PROPERTY ModuloTurn : dint
GET
ModuloTurn := _Mover.NcToPlc.ModuloSetTurns;
END_GET
END_PROPERTY

PROPERTY Mover : REFERENCE to AXIS_REF
SET
_Mover REF= Mover;
END_SET
END_PROPERTY

PROPERTY MoverId : uint
SET
_nMoverId := MoverId;
END_SET
END_PROPERTY

PROPERTY MoverInfo : REFERENCE to ST_MOVER_INFO
SET


	_stInfo ref= MoverInfo;
END_SET
END_PROPERTY

METHOD MoveToPos : E_PROGRESS
VAR_INPUT
  Execute             : BOOL;
  stMoveData          : ST_MOVE_DATA;
END_VAR
VAR_INST
  _nErrorId           : UDINT;
  _rDelta,
  _rPos               : LREAL;
  _eState             : E_PROGRESS;
END_VAR
IF NOT Execute THEN _eState  := E_PROGRESS.PROGRESS_INIT; END_IF 
IF NOT Check() THEN MoveToPos   := E_PROGRESS.PROGRESS_ERROR; RETURN; END_IF


CASE _eState
OF
  E_PROGRESS.PROGRESS_INIT:
    IF Execute
    THEN
      _nErrorId               := 0;
      _rDelta                 := SEL((stMoveData.rDelta < 0.01), stMoveData.rDelta, 0.05);
      _eState                 := E_PROGRESS.PROGRESS_BUSY;
    END_IF
END_CASE
//-----------------------------------------------------------------------------
//-----------------------------------------------------------------------------
CASE _eState
OF
  E_PROGRESS.PROGRESS_BUSY:
    _eState                   := E_PROGRESS.PROGRESS_PREPARE;
    _fbPower.Override         := stMoveData.rOverride;

    _rPos                     := ABS(_Mover.NcToPlc.ModuloActTurns)* _RailLength + stMoveData.rPos;


    _rLastPosition            := _rPos;
    //_rLastGap                 := stMoveData.rGap;

    _fbMoveAbs(
            Axis              := _Mover, 
            Execute           := FALSE, 
            Position          := _rPos, 
            Velocity          := stMoveData.rVelo, 
            Acceleration      := stMoveData.rAcc, 
            Deceleration      := stMoveData.rAcc, 
            Jerk              := stMoveData.rJerk, 
            BufferMode        := Tc2_MC2.MC_BufferMode.MC_Aborting);

      IF (_eMessageLevel > E_MessageType.eMessageInfo)
      THEN
        _stMsg.eType          := E_MessageType.eMessageVerbose;
        _stMsg.eSubdevice     := e_Subdevice.fbMovePtP;
        _stMsg.iErrorNumber   := _nErrorId;
        _stMsg.sText          := concat(TO_STRING(_eState), ': ');
        _stMsg.sText          := concat(_stMsg.sText, concat('stMoveData.rPos: ', TO_STRING(stMoveData.rPos)));
        f_MessageSet(_stMsg);
      END_IF
END_CASE
//-----------------------------------------------------------------------------
//-----------------------------------------------------------------------------
CASE _eState
OF
  E_PROGRESS.PROGRESS_PREPARE:
    _fbMoveAbs(
            Axis              := _Mover, 
            Execute           := TRUE, 
            Position          := _rPos, 
            Velocity          := stMoveData.rVelo, 
            Acceleration      := stMoveData.rAcc, 
            Deceleration      := stMoveData.rAcc, 
            Jerk              := stMoveData.rJerk, 
            BufferMode        := Tc2_MC2.MC_BufferMode.MC_Aborting);

    IF _fbMoveAbs.Error
    THEN
      _bError                 := TRUE;
      _nErrorId               := _fbMoveAbs.ErrorId;
      _eState                 := E_PROGRESS.PROGRESS_ERROR;

      _stMsg.eType            := E_MessageType.eMessageError;
      _stMsg.eSubdevice       := e_Subdevice.fbMovePtP;
      _stMsg.iErrorNumber     := _nErrorId;
      _stMsg.sText            := TO_STRING(_eState);
      f_MessageSet(_stMsg);

    ELSIF _fbMoveAbs.Active OR 
          _fbMoveAbs.Done
		THEN
      _eState                 := E_PROGRESS.PROGRESS_WORKING;

      IF (_eMessageLevel = E_MessageType.eMessageVerbose)
      THEN
        _stMsg.eType          := E_MessageType.eMessageVerbose;
        _stMsg.eSubdevice     := e_Subdevice.fbMovePtP;
        _stMsg.iErrorNumber   := _nErrorId;
        _stMsg.sText          := concat(TO_STRING(_eState), ': ');
        _stMsg.sText          := concat(_stMsg.sText, '.ModuloActPos: ');
        _stMsg.sText          := concat(_stMsg.sText, TO_STRING(_Mover.NcToPlc.ModuloActPos));
        f_MessageSet(_stMsg);
      END_IF
    END_IF
END_CASE
//-----------------------------------------------------------------------------
//-----------------------------------------------------------------------------
CASE _eState
OF
  E_PROGRESS.PROGRESS_WORKING:
    _fbMoveAbs(
          Axis                := _Mover);

    IF _fbMoveAbs.Error
    THEN
      _bError                 := TRUE;
      _nErrorId               := _fbMoveAbs.ErrorId;
      _stInfo.nErrorId        := _nErrorId;
      _eState                 := E_PROGRESS.PROGRESS_ERROR;

      _stMsg.eType            := E_MessageType.eMessageError;
      _stMsg.eSubdevice       := e_Subdevice.fbMovePtP;
      _stMsg.iErrorNumber     := _nErrorId;
      _stMsg.sText            := TO_STRING(_eState);
      f_MessageSet(_stMsg);

      _fbMoveAbs( 
            Axis              := _Mover, 
            Execute           := FALSE);


    ELSIF (_Mover.NcToPlc.ActPos > _fbMoveAbs.Position - _rDelta) AND
          (_Mover.NcToPlc.ActPos < _fbMoveAbs.Position + _rDelta)
    THEN
      IF NOT _Mover.Status.Moving
      THEN
        _eState               := E_PROGRESS.PROGRESS_DONE;

        IF (_eMessageLevel > E_MessageType.eMessageError)
        THEN
          _stMsg.eType        := E_MessageType.eMessageInfo;
          _stMsg.eSubdevice   := e_Subdevice.fbMovePtP;
          _stMsg.iErrorNumber := _nErrorId;
          _stMsg.sText        := concat(TO_STRING(_eState), ': ');
          _stMsg.sText        := concat(_stMsg.sText, concat('ModActPos: ', TO_STRING(_Mover.NcToPlc.ModuloActPos)));
          f_MessageSet(_stMsg);
        END_IF
      _fbMoveAbs( 
            Axis              := _Mover, 
            Execute           := FALSE);
      END_IF
    END_IF
END_CASE
//-----------------------------------------------------------------------------
//-----------------------------------------------------------------------------

MoveToPos                   := _eState;
END_METHOD

METHOD MoveToPosCa : E_PROGRESS
VAR_INPUT
  Execute             : BOOL;
  stMoveData          : ST_MOVE_DATA;
END_VAR
VAR_INST
  _nErrorId           : UDINT;
  _rDelta,
  _rPos               : LREAL;
  _eState             : E_PROGRESS;
END_VAR
IF NOT Execute THEN _eState  := E_PROGRESS.PROGRESS_INIT; END_IF 
IF NOT Check() THEN MoveToPosCa   := E_PROGRESS.PROGRESS_ERROR; RETURN; END_IF


CASE _eState
OF
  E_PROGRESS.PROGRESS_INIT:
    IF Execute
    THEN
      _nErrorId               := 0;
      _rDelta                 := SEL((stMoveData.rDelta < 0.01), stMoveData.rDelta, 0.05);
      _eState                 := E_PROGRESS.PROGRESS_BUSY;
    END_IF
END_CASE
//-----------------------------------------------------------------------------
//-----------------------------------------------------------------------------
CASE _eState
OF
  E_PROGRESS.PROGRESS_BUSY:
    _eState                   := E_PROGRESS.PROGRESS_PREPARE;
    _fbPower.Override         := stMoveData.rOverride;

    _rPos                     := ABS(_Mover.NcToPlc.ModuloActTurns)* _RailLength + stMoveData.rPos;


    _rLastPosition            := _rPos;
    _rLastGap                 := stMoveData.rGap;

    _fbMoveAbsCa( 
            Axis              := _Mover, 
            Execute           := FALSE, 
            ContinuousUpdate  := TRUE, 
            Position          := _rPos,
            Velocity          := stMoveData.rVelo, 
            Acceleration      := stMoveData.rAcc, 
            Deceleration      := stMoveData.rAcc, 
            Jerk              := stMoveData.rJerk, 
            Gap               := stMoveData.rGap, 
            BufferMode        := Tc3_Mc3Definitions.MC_BUFFER_MODE.mcAborting);

    IF (_eMessageLevel > E_MessageType.eMessageInfo)
    THEN
      _stMsg.eType            := E_MessageType.eMessageVerbose;
      _stMsg.eSubdevice       := e_Subdevice.fbMoveToPosCa;
      _stMsg.iErrorNumber     := _nErrorId;
      _stMsg.sText            := concat(TO_STRING(_eState), ': ');
      _stMsg.sText            := concat(_stMsg.sText, concat('stMoveData.rPos: ', TO_STRING(stMoveData.rPos)));
      f_MessageSet(_stMsg);
    END_IF
END_CASE
//-----------------------------------------------------------------------------
//-----------------------------------------------------------------------------
CASE _eState
OF
  E_PROGRESS.PROGRESS_PREPARE:
    _fbMoveAbsCa( 
            Axis              := _Mover, 
            Execute           := TRUE, 
            ContinuousUpdate  := TRUE, 
            Position          := _rPos,
            Velocity          := stMoveData.rVelo, 
            Acceleration      := stMoveData.rAcc, 
            Deceleration      := stMoveData.rAcc, 
            Jerk              := stMoveData.rJerk, 
            Gap               := stMoveData.rGap, 
            BufferMode        := Tc3_Mc3Definitions.MC_BUFFER_MODE.mcAborting);

    IF _fbMoveAbsCa.Error
    THEN
      _bError                 := TRUE;
      _nErrorId               := _fbMoveAbsCa.ErrorId;
      _stInfo.nErrorId        := _nErrorId;
      _eState                 := E_PROGRESS.PROGRESS_ERROR;

      _stMsg.eType            := E_MessageType.eMessageError;
      _stMsg.eSubdevice       := e_Subdevice.fbMoveToPosCa;
      _stMsg.iErrorNumber     := _nErrorId;
      _stMsg.sText            := TO_STRING(_eState);
      f_MessageSet(_stMsg);

    ELSIF _fbMoveAbsCa.Active OR 
          _fbMoveAbsCa.Done
		THEN
      _eState                 := E_PROGRESS.PROGRESS_WORKING;

      IF (_eMessageLevel = E_MessageType.eMessageVerbose)
      THEN
        _stMsg.eType          := E_MessageType.eMessageVerbose;
        _stMsg.eSubdevice     := e_Subdevice.fbMoveToPosCa;
        _stMsg.iErrorNumber   := _nErrorId;
        _stMsg.sText          := concat(TO_STRING(_eState), ': ');
        _stMsg.sText          := concat(_stMsg.sText, '.ModuloActPos: ');
        _stMsg.sText          := concat(_stMsg.sText, TO_STRING(_Mover.NcToPlc.ModuloActPos));
        f_MessageSet(_stMsg);
      END_IF
    END_IF
END_CASE
//-----------------------------------------------------------------------------
//-----------------------------------------------------------------------------
CASE _eState
OF
  E_PROGRESS.PROGRESS_WORKING:
    _fbMoveAbsCa(
          Axis                := _Mover);

    IF _fbMoveAbsCa.Error
    THEN
      _bError                 := TRUE;
      _nErrorId               := _fbMoveAbsCa.ErrorId;
      _stInfo.nErrorId        := _nErrorId;
      _fbMoveAbsCa( 
            Axis              := _Mover, 
            Execute           := FALSE);

      _eState                 := E_PROGRESS.PROGRESS_ERROR;

      _stMsg.eType            := E_MessageType.eMessageError;
      _stMsg.eSubdevice       := e_Subdevice.fbMoveToPosCa;
      _stMsg.iErrorNumber     := _nErrorId;
      _stMsg.sText            := concat(TO_STRING(_eState), ': ');
      _stMsg.sText            := concat(_stMsg.sText, concat('ModActPos: ', TO_STRING(_Mover.NcToPlc.ModuloActPos)));

      f_MessageSet(_stMsg);

    ELSIF (_Mover.NcToPlc.ActPos > _fbMoveAbsCa.Position - _rDelta) AND
          (_Mover.NcToPlc.ActPos < _fbMoveAbsCa.Position + _rDelta)
    THEN
      IF NOT _Mover.Status.Moving
      THEN
        _eState               := E_PROGRESS.PROGRESS_DONE;

        IF (_eMessageLevel > E_MessageType.eMessageError)
        THEN
          _stMsg.eType        := E_MessageType.eMessageInfo;
          _stMsg.eSubdevice   := e_Subdevice.fbMoveToPosCa;
          _stMsg.iErrorNumber := _nErrorId;
          _stMsg.sText        := concat(TO_STRING(_eState), ': ');
          _stMsg.sText        := concat(_stMsg.sText, concat('ModActPos: ', TO_STRING(_Mover.NcToPlc.ModuloActPos)));
          f_MessageSet(_stMsg);
        END_IF
      _fbMoveAbsCa( 
            Axis              := _Mover, 
            Execute           := FALSE);
      END_IF
    END_IF
END_CASE
//-----------------------------------------------------------------------------
//-----------------------------------------------------------------------------

MoveToPosCa                   := _eState;
END_METHOD

PROPERTY RailLength : LREAL
GET
RailLength := _RailLength;
END_GET
SET
_RailLength := RailLength;
END_SET
END_PROPERTY

METHOD Reset : E_PROGRESS
VAR_INPUT
  Execute             : BOOL;
END_VAR
VAR_INST
  _nErrorId           : UDINT;
  _eState             : E_PROGRESS;
END_VAR
IF NOT Execute THEN _eState  := E_PROGRESS.PROGRESS_INIT; END_IF 
IF NOT Check() THEN Reset    := E_PROGRESS.PROGRESS_ERROR; RETURN; END_IF


CASE _eState
OF
  E_PROGRESS.PROGRESS_INIT:
    IF Execute
    THEN
      _stInfo.nErrorId        :=
      _nErrorId               := 0;
      _eState                 := E_PROGRESS.PROGRESS_BUSY;
    END_IF
END_CASE
//-----------------------------------------------------------------------------
//-----------------------------------------------------------------------------
CASE _eState
OF
  E_PROGRESS.PROGRESS_BUSY:
    _eState                   := E_PROGRESS.PROGRESS_PREPARE;
    _fbReset(
            Axis              := _Mover, 
            Execute           := FALSE);

    IF (_eMessageLevel > E_MessageType.eMessageInfo)
    THEN
      _stMsg.eType            := E_MessageType.eMessageVerbose;
      _stMsg.eSubdevice       := e_Subdevice.fbReset;
      _stMsg.iErrorNumber     := _nErrorId;
      _stMsg.sText            := TO_STRING(_eState);
      f_MessageSet(_stMsg);
    END_IF
END_CASE
//-----------------------------------------------------------------------------
//-----------------------------------------------------------------------------
CASE _eState
OF
  E_PROGRESS.PROGRESS_PREPARE:
    _fbReset(
            Axis              := _Mover, 
            Execute           := TRUE);

    IF _fbReset.Error
    THEN
      _nErrorId               := _fbReset.ErrorID;
      _eState                 := E_PROGRESS.PROGRESS_ERROR;

      _stMsg.eType            := E_MessageType.eMessageError;
      _stMsg.eSubdevice       := e_Subdevice.fbReset;
      _stMsg.iErrorNumber     := _nErrorId;
      _stMsg.sText            := TO_STRING(_eState);
      f_MessageSet(_stMsg);

    ELSIF NOT _Mover.Status.Moving
    THEN
      _eState                 := E_PROGRESS.PROGRESS_DONE;

      IF (_eMessageLevel > E_MessageType.eMessageError)
      THEN
        _stMsg.eType          := E_MessageType.eMessageInfo;
        _stMsg.eSubdevice     := e_Subdevice.fbReset;
        _stMsg.iErrorNumber   := _nErrorId;
        _stMsg.sText          := TO_STRING(_eState);
        f_MessageSet(_stMsg);
      END_IF
    END_IF
END_CASE
//-----------------------------------------------------------------------------
//-----------------------------------------------------------------------------
CASE _eState
OF
  E_PROGRESS.PROGRESS_ERROR,
  E_PROGRESS.PROGRESS_DONE:
    _stInfo.nErrorId          := _nErrorId;
    _fbReset(
            Axis              := _Mover, 
            Execute           := FALSE);
			
	_bError := FALSE;		
END_CASE
//-----------------------------------------------------------------------------
//-----------------------------------------------------------------------------

Reset                         := _eState;
END_METHOD

METHOD SendToAbsPosCa : E_PROGRESS
VAR_INPUT
  Execute             : BOOL;
  stMoveData          : ST_MOVE_DATA;
END_VAR
VAR_INST
  _nErrorId           : UDINT;
  _rPos               : LREAL;
  _rStart             : LREAL;
  _eState             : E_PROGRESS;
END_VAR
IF NOT Execute THEN _eState  := E_PROGRESS.PROGRESS_INIT; END_IF 
IF NOT Check() THEN SendToAbsPosCa   := E_PROGRESS.PROGRESS_ERROR; RETURN; END_IF


CASE _eState
OF
  E_PROGRESS.PROGRESS_INIT:
    IF Execute
    THEN
      _nErrorId               := 0;
      _rStart                 := _Mover.NcToPlc.ActPos;

      _eState                 := E_PROGRESS.PROGRESS_BUSY;
    END_IF
END_CASE
//-----------------------------------------------------------------------------
//-----------------------------------------------------------------------------
CASE _eState
OF
  E_PROGRESS.PROGRESS_BUSY:
    _eState                   := E_PROGRESS.PROGRESS_PREPARE;
    _fbPower.Override         := stMoveData.rOverride;

    _rPos                     := stMoveData.rPos;
	
    _rLastPosition            := _rPos;
    _rLastGap                 := stMoveData.rGap;

    _fbMoveAbsCa( 
            Axis              := _Mover, 
            Execute           := FALSE, 
            ContinuousUpdate  := TRUE, 
            Position          := _rPos,
            Velocity          := stMoveData.rVelo, 
            Acceleration      := stMoveData.rAcc, 
            Deceleration      := stMoveData.rAcc, 
            Jerk              := stMoveData.rJerk, 
            Gap               := stMoveData.rGap, 
            BufferMode        := Tc3_Mc3Definitions.MC_BUFFER_MODE.mcAborting);

    IF (_eMessageLevel > E_MessageType.eMessageVerbose)
    THEN
      _stMsg.eType            := E_MessageType.eMessageSentient;
      _stMsg.eSubdevice       := e_Subdevice.fbSendToAbsPosCa;
      _stMsg.iErrorNumber     := _nErrorId;
      _stMsg.sText            := concat(TO_STRING(_eState), ': ');
      _stMsg.sText            := concat(_stMsg.sText, 'stMoveData.rPos: ');
      _stMsg.sText            := concat(_stMsg.sText, TO_STRING(stMoveData.rPos));
      f_MessageSet(_stMsg);

      _stMsg.eType            := E_MessageType.eMessageSentient;
      _stMsg.eSubdevice       := e_Subdevice.fbSendToAbsPosCa;
      _stMsg.iErrorNumber     := _nErrorId;
      _stMsg.sText            := concat(TO_STRING(_eState), ': ');
      _stMsg.sText            := concat(_stMsg.sText, '.rDistance: ');
      _stMsg.sText            := concat(_stMsg.sText, TO_STRING(stMoveData.rDistance));
      f_MessageSet(_stMsg);
    END_IF
END_CASE
//-----------------------------------------------------------------------------
//-----------------------------------------------------------------------------
CASE _eState
OF
  E_PROGRESS.PROGRESS_PREPARE:
    _fbMoveAbsCa( 
            Axis              := _Mover, 
            Execute           := TRUE, 
            ContinuousUpdate  := TRUE, 
            Position          := _rPos,
            Velocity          := stMoveData.rVelo, 
            Acceleration      := stMoveData.rAcc, 
            Deceleration      := stMoveData.rAcc, 
            Jerk              := stMoveData.rJerk, 
            Gap               := stMoveData.rGap, 
            BufferMode        := Tc3_Mc3Definitions.MC_BUFFER_MODE.mcAborting);

    IF _fbMoveAbsCa.Error
    THEN
      _bError                 := TRUE;
      _nErrorId               := _fbMoveAbsCa.ErrorId;
      _stInfo.nErrorId        := _nErrorId;
      _eState                 := E_PROGRESS.PROGRESS_ERROR;

      _stMsg.eType            := E_MessageType.eMessageError;
      _stMsg.eSubdevice       := e_Subdevice.fbSendToAbsPosCa;
      _stMsg.iErrorNumber     := _nErrorId;
      _stMsg.sText            := TO_STRING(_eState);
      f_MessageSet(_stMsg);

    ELSIF _fbMoveAbsCa.Active OR
          _fbMoveAbsCa.Done
    THEN
      _eState                 := E_PROGRESS.PROGRESS_WORKING;

      IF (_eMessageLevel > E_MessageType.eMessageVerbose)
      THEN
        _stMsg.eType          := E_MessageType.eMessageSentient;
        _stMsg.eSubdevice     := e_Subdevice.fbSendToAbsPosCa;
        _stMsg.iErrorNumber   := _nErrorId;
        _stMsg.sText          := concat(TO_STRING(_eState), ': ');
        _stMsg.sText          := concat(_stMsg.sText, '.ActPos: ');
        _stMsg.sText          := concat(_stMsg.sText, TO_STRING(_Mover.NcToPlc.ActPos));
        //f_MessageSet(_stMsg);
      END_IF
    END_IF
END_CASE
//-----------------------------------------------------------------------------
//-----------------------------------------------------------------------------
CASE _eState
OF
  E_PROGRESS.PROGRESS_WORKING:
    _fbMoveAbsCa(
            Axis              := _Mover);

    IF _fbMoveAbsCa.Error
    THEN
      _bError                 := TRUE;
      _nErrorId               := _fbMoveAbsCa.ErrorId;
      _stInfo.nErrorId        := _nErrorId;
      _fbMoveAbsCa( 
            Axis              := _Mover, 
            Execute           := FALSE);

      _eState                 := E_PROGRESS.PROGRESS_ERROR;

      _stMsg.eType            := E_MessageType.eMessageError;
      _stMsg.eSubdevice       := e_Subdevice.fbSendToAbsPosCa;
      _stMsg.iErrorNumber     := _nErrorId;
      _stMsg.sText            := TO_STRING(_eState);
      f_MessageSet(_stMsg);

    ELSIF (_Mover.NcToPlc.ActPos > _rStart + stMoveData.rDistance)
    THEN
      _eState                 := E_PROGRESS.PROGRESS_DONE;

      IF (_eMessageLevel > E_MessageType.eMessageError)
      THEN
        _stMsg.eType          := E_MessageType.eMessageInfo;
        _stMsg.eSubdevice     := e_Subdevice.fbSendToAbsPosCa;
        _stMsg.iErrorNumber   := _nErrorId;
        _stMsg.sText          := concat(TO_STRING(_eState), ': ');
        _stMsg.sText          := concat(_stMsg.sText, '.ActPos: ');
        _stMsg.sText          := concat(_stMsg.sText, TO_STRING(_Mover.NcToPlc.ActPos));
        _stMsg.sText          := concat(_stMsg.sText, ' ');
        _stMsg.sText          := concat(_stMsg.sText, '.ActVelo: ');
        _stMsg.sText          := concat(_stMsg.sText, TO_STRING(_Mover.NcToPlc.ActVelo));

        f_MessageSet(_stMsg);
      END_IF
      _fbMoveAbsCa( 
            Axis              := _Mover, 
            Execute           := FALSE);
    END_IF
END_CASE
//-----------------------------------------------------------------------------
//-----------------------------------------------------------------------------

SendToAbsPosCa                := _eState;
END_METHOD

METHOD SendToModuloPosCa : E_PROGRESS
VAR_INPUT
  Execute             : BOOL;
  stMoveData          : ST_MOVE_DATA;
END_VAR
VAR_INST
  _nErrorId           : UDINT;
  _rPos               : LREAL;
  _rStart             : LREAL;
  _eState             : E_PROGRESS;
END_VAR
IF NOT Execute THEN _eState  := E_PROGRESS.PROGRESS_INIT; END_IF 
IF NOT Check() THEN SendToModuloPosCa   := E_PROGRESS.PROGRESS_ERROR; RETURN; END_IF


CASE _eState
OF
  E_PROGRESS.PROGRESS_INIT:
    IF Execute
    THEN
      _nErrorId               := 0;
      _rStart                 := _Mover.NcToPlc.ActPos;

      _eState                 := E_PROGRESS.PROGRESS_BUSY;
    END_IF
    _fbMoveAbsCa( 
          Axis              := _Mover, 
          Execute           := FALSE);
END_CASE
//-----------------------------------------------------------------------------
//-----------------------------------------------------------------------------
CASE _eState
OF
  E_PROGRESS.PROGRESS_BUSY:
    _eState                   := E_PROGRESS.PROGRESS_PREPARE;
    _fbPower.Override         := stMoveData.rOverride;

    _rPos                     := ABS(_Mover.NcToPlc.ModuloActTurns)* _RailLength + stMoveData.rPos;
	
    _rLastPosition            := _rPos;
    _rLastGap                 := stMoveData.rGap;

    _fbMoveAbsCa( 
            Axis              := _Mover, 
            Execute           := FALSE, 
            ContinuousUpdate  := TRUE, 
            Position          := _rPos,
            Velocity          := stMoveData.rVelo, 
            Acceleration      := stMoveData.rAcc, 
            Deceleration      := stMoveData.rAcc, 
            Jerk              := stMoveData.rJerk, 
            Gap               := stMoveData.rGap, 
            BufferMode        := Tc3_Mc3Definitions.MC_BUFFER_MODE.mcAborting);

    IF (_eMessageLevel > E_MessageType.eMessageVerbose)
    THEN
      _stMsg.eType            := E_MessageType.eMessageSentient;
      _stMsg.eSubdevice       := e_Subdevice.fbSendToModuloPosCa;
      _stMsg.iErrorNumber     := _nErrorId;
      _stMsg.sText            := concat(TO_STRING(_eState), ': ');
      _stMsg.sText            := concat(_stMsg.sText, 'stMoveData.rPos: ');
      _stMsg.sText            := concat(_stMsg.sText, TO_STRING(stMoveData.rPos));
      f_MessageSet(_stMsg);

      _stMsg.eType            := E_MessageType.eMessageSentient;
      _stMsg.eSubdevice       := e_Subdevice.fbSendToModuloPosCa;
      _stMsg.iErrorNumber     := _nErrorId;
      _stMsg.sText            := concat(TO_STRING(_eState), ': ');
      _stMsg.sText            := concat(_stMsg.sText, '.rDistance: ');
      _stMsg.sText            := concat(_stMsg.sText, TO_STRING(stMoveData.rDistance));
      f_MessageSet(_stMsg);

    END_IF
END_CASE
//-----------------------------------------------------------------------------
//-----------------------------------------------------------------------------
CASE _eState
OF
  E_PROGRESS.PROGRESS_PREPARE:
    _fbMoveAbsCa( 
            Axis              := _Mover, 
            Execute           := TRUE, 
            ContinuousUpdate  := TRUE, 
            Position          := _rPos,
            Velocity          := stMoveData.rVelo, 
            Acceleration      := stMoveData.rAcc, 
            Deceleration      := stMoveData.rAcc, 
            Jerk              := stMoveData.rJerk, 
            Gap               := stMoveData.rGap, 
            BufferMode        := Tc3_Mc3Definitions.MC_BUFFER_MODE.mcAborting);

    IF _fbMoveAbsCa.Error
    THEN
      _bError                 := TRUE;
      _nErrorId               := _fbMoveAbsCa.ErrorId;
      _stInfo.nErrorId        := _nErrorId;
      _eState                 := E_PROGRESS.PROGRESS_ERROR;

      _stMsg.eType            := E_MessageType.eMessageError;
      _stMsg.eSubdevice       := e_Subdevice.fbSendToModuloPosCa;
      _stMsg.iErrorNumber     := _nErrorId;
      _stMsg.sText            := TO_STRING(_eState);
      f_MessageSet(_stMsg);

      _fbMoveAbsCa( 
            Axis              := _Mover, 
            Execute           := FALSE);

    ELSIF _fbMoveAbsCa.Active OR
          _fbMoveAbsCa.Done
    THEN
      _eState                 := E_PROGRESS.PROGRESS_WORKING;

      IF (_eMessageLevel > E_MessageType.eMessageVerbose)
      THEN
        _stMsg.eType          := E_MessageType.eMessageSentient;
        _stMsg.eSubdevice     := e_Subdevice.fbSendToModuloPosCa;
        _stMsg.iErrorNumber   := _nErrorId;
        _stMsg.sText            := concat(TO_STRING(_eState), ': ');
        _stMsg.sText          := concat(_stMsg.sText, '.ModuloActPos: ');
        _stMsg.sText          := concat(_stMsg.sText, TO_STRING(_Mover.NcToPlc.ModuloActPos));
        //f_MessageSet(_stMsg);
      END_IF
(*
    ELSIF (_Mover.NcToPlc.ActPos > _rStart + stMoveData.rDistance)
    THEN
      _eState                 := E_PROGRESS.PROGRESS_DONE;

      IF (_eMessageLevel < E_MessageType.eMessageError)
      THEN
        _stMsg.eType          := E_MessageType.eMessageInfo;
        _stMsg.eSubdevice     := e_Subdevice.fbSendToModuloPosCa;
        _stMsg.iErrorNumber   := _nErrorId;
        _stMsg.sText          := TO_STRING(_eState);
        f_MessageSet(_stMsg);
      END_IF
      _fbMoveAbsCa( 
            Axis              := _Mover, 
            Execute           := FALSE);
*)
    END_IF
END_CASE
//-----------------------------------------------------------------------------
//-----------------------------------------------------------------------------
CASE _eState
OF
  E_PROGRESS.PROGRESS_WORKING:
    _fbMoveAbsCa(
            Axis              := _Mover);

    IF _fbMoveAbsCa.Error
    THEN
      _bError                 := TRUE;
      _nErrorId               := _fbMoveAbsCa.ErrorId;
      _stInfo.nErrorId        := _nErrorId;
      _fbMoveAbsCa( 
            Axis              := _Mover, 
            Execute           := FALSE);

      _eState                 := E_PROGRESS.PROGRESS_ERROR;

      _stMsg.eType            := E_MessageType.eMessageError;
      _stMsg.eSubdevice       := e_Subdevice.fbSendToModuloPosCa;
      _stMsg.iErrorNumber     := _nErrorId;
      _stMsg.sText            := TO_STRING(_eState);
      f_MessageSet(_stMsg);

    ELSIF (_Mover.NcToPlc.ActPos > _rStart + stMoveData.rDistance)
    THEN
      _eState                 := E_PROGRESS.PROGRESS_DONE;

      IF (_eMessageLevel > E_MessageType.eMessageError)
      THEN
        _stMsg.eType          := E_MessageType.eMessageInfo;
        _stMsg.eSubdevice     := e_Subdevice.fbSendToModuloPosCa;
        _stMsg.iErrorNumber   := _nErrorId;
        _stMsg.sText          := concat(TO_STRING(_eState), ': ');
        _stMsg.sText          := concat(_stMsg.sText, '.ModuloActPos: ');
        _stMsg.sText          := concat(_stMsg.sText, TO_STRING(_Mover.NcToPlc.ModuloActPos));
        _stMsg.sText          := concat(_stMsg.sText, ' ');
        _stMsg.sText          := concat(_stMsg.sText, '.ActVelo: ');
        _stMsg.sText          := concat(_stMsg.sText, TO_STRING(_Mover.NcToPlc.ActVelo));
        f_MessageSet(_stMsg);
      END_IF
      _fbMoveAbsCa( 
            Axis              := _Mover, 
            Execute           := FALSE);
    END_IF
END_CASE
//-----------------------------------------------------------------------------
//-----------------------------------------------------------------------------

SendToModuloPosCa                   := _eState;
END_METHOD

METHOD Stop : E_PROGRESS
VAR_INPUT
  Execute             : BOOL;
  stMoveData          : ST_MOVE_DATA;
END_VAR
VAR_INST
  _nErrorId           : UDINT;
  _eState             : E_PROGRESS;
END_VAR
IF NOT Execute 
THEN 
	_eState := E_PROGRESS.PROGRESS_INIT; 
END_IF 
IF NOT Check() 
THEN 
	Stop := E_PROGRESS.PROGRESS_ERROR; 
	RETURN; 
END_IF


CASE _eState
OF
  E_PROGRESS.PROGRESS_INIT:
    IF Execute
    THEN
      _nErrorId               := 0;
      _eState                 := E_PROGRESS.PROGRESS_BUSY;
    END_IF
END_CASE
//-----------------------------------------------------------------------------
//-----------------------------------------------------------------------------
CASE _eState
OF
  E_PROGRESS.PROGRESS_BUSY:
    _eState                   := E_PROGRESS.PROGRESS_PREPARE;
    _fbStop(
            Axis              := _Mover, 
            Execute           := FALSE, 
            Deceleration      := stMoveData.rAcc, 
            Jerk              := stMoveData.rJerk); 

    IF (_eMessageLevel > E_MessageType.eMessageInfo)
    THEN
      _stMsg.eType            := E_MessageType.eMessageVerbose;
      _stMsg.eSubdevice       := e_Subdevice.fbStop;
      _stMsg.iErrorNumber     := _nErrorId;
      _stMsg.sText            := TO_STRING(_eState);
      f_MessageSet(_stMsg);
    END_IF
END_CASE
//-----------------------------------------------------------------------------
//-----------------------------------------------------------------------------
CASE _eState
OF
  E_PROGRESS.PROGRESS_PREPARE:
    _fbStop(Axis              := _Mover, 
            Execute           := TRUE, 
            Deceleration      := stMoveData.rAcc, 
            Jerk              := stMoveData.rJerk);

    IF _fbStop.Error
    THEN
      _bError                 := TRUE;
      _nErrorId               := _fbStop.ErrorID;
      _eState                 := E_PROGRESS.PROGRESS_ERROR;

      _stMsg.eType            := E_MessageType.eMessageError;
      _stMsg.eSubdevice       := e_Subdevice.fbStop;
      _stMsg.iErrorNumber     := _nErrorId;
      _stMsg.sText            := TO_STRING(_eState);
      f_MessageSet(_stMsg);

    ELSIF _fbStop.Done
    THEN
      _eState                 := E_PROGRESS.PROGRESS_DONE;

      IF (_eMessageLevel > E_MessageType.eMessageError)
      THEN
        _stMsg.eType          := E_MessageType.eMessageInfo;
        _stMsg.eSubdevice     := e_Subdevice.fbStop;
        _stMsg.iErrorNumber   := _nErrorId;
        _stMsg.sText          := TO_STRING(_eState);
        f_MessageSet(_stMsg);
      END_IF
    END_IF
END_CASE
//-----------------------------------------------------------------------------
//-----------------------------------------------------------------------------
CASE _eState
OF
  E_PROGRESS.PROGRESS_ERROR,
  E_PROGRESS.PROGRESS_DONE:
    _stInfo.nErrorId          := _nErrorId;
    _fbStop(
            Axis              := _Mover, 
            Execute           := FALSE);
END_CASE
//-----------------------------------------------------------------------------
//-----------------------------------------------------------------------------

Stop                          := _eState;
END_METHOD

END_FUNCTION_BLOCK

// ---- APPLICATION/_types/Initialization_Robot.TcPOU
FUNCTION Initialization_Robot : BOOL
VAR_INPUT
END_VAR
VAR
  _nBufferOutfeedTarget       : ARRAY[1..2] OF E_INSTANCE;
  _nStnFrst                   : UINT;
END_VAR

//*************************************************************************************************************
//
// build configuration for Instances and ProcessInterfaces
//
//*************************************************************************************************************
//*************************************************************************************************************
// - ProcessConductor : Instance with connection to a cyclic linked list 
//                      Here does The Ticket with target processId and bitmask arrive 
//                      this instance forwards the ticket to its destination
//                        destination is BufferInfeed
//-------------------------------------------------------------------------------------------------------------
// whoami
//
// ticket box - transfersystem drops ticket
//-------------------------------------------------------------------------------------------------------------
ProcessConductor.ProcessId                := ProcessCollector[E_INSTANCE.PROCESS_CONDUCTOR].ProcessId;
ProcessConductor.CollectorInterface       := ItfProcessCollector;
ProcessConductor.ProcessLinkedLists       := ItfProcessList;

//*************************************************************************************************************
// - BufferInfeed     : single XtsStation which looks for input trigger from transfersystem, 
//                      transfersystem writes positions of XtsStations to be used at Infeed. 
//                      BufferInfeed is writing ItfProcessCollector[BufferInfeed.ProcessTarget].ActivateStation 
//                        for BufferInfeed target (Infeed / 12 XtsStations).
//                      BufferInfeed sends required amount of movers to WaitPos of XtsStations 
//                        of BufferInfeed target (Infeed / 12 XtsStations).
//-------------------------------------------------------------------------------------------------------------
// whoami
//
// process target (Infeed / 12 XtsStations)
//-------------------------------------------------------------------------------------------------------------
BufferInfeed.ProcessId                    := ProcessCollector[E_INSTANCE.BUFFER_INFEED].ProcessId;
BufferInfeed.ProcessTarget                := ProcessCollector[E_INSTANCE.INFEED].ProcessId;
BufferInfeed.CollectorInterface           := ItfProcessCollector;
BufferInfeed.ProcessLinkedLists           := ItfProcessList;
//-------------------------------------------------------------------------------------------------------------
// configure range of XtsStations for process
//
// see MAIN.StationParameterInit() for positions and dyn constraints
//-------------------------------------------------------------------------------------------------------------
ItfProcessCollector[BufferInfeed.ProcessId].StationFirst  := 53;
ItfProcessCollector[BufferInfeed.ProcessId].StationLast   := 53;

_nStnFrst                                 := ProcessCollector[BufferInfeed.ProcessId].StationFirst;
BufferInfeed.CheckPosition                := 15.0;

//-------------------------------------------------------------------------------------------------------------
//-------------------------------------------------------------------------------------------------------------
//*************************************************************************************************************
//*************************************************************************************************************
// - Infeed         : 12 XtsStations for transfersystem to unload
//                    Infeed is pulling in the movers according to list entry from BufferInfeed
//                    one stop only
//                    must be checked for all mover standstill in PosStop[1] of each XtsStation
//                    must be released by handshake from transfersystem (this is done by a TON for now)
//-------------------------------------------------------------------------------------------------------------
// whoami
//
// process target (BufferOutfeed / 1 XtsStation)
// TODO: 
//    configure infeed target for OUTFEED_CLAMP (12 XtsStations)
//    Infeed.ProcessTarget  := ProcessCollector[E_INSTANCE.OUTFEED_CLAMP].ProcessId;
//-------------------------------------------------------------------------------------------------------------
Infeed.ProcessId                          := ProcessCollector[E_INSTANCE.INFEED].ProcessId;
Infeed.ProcessTarget                      := ProcessCollector[E_INSTANCE.BUFFER_OUTFEED].ProcessId;
Infeed.CollectorInterface                 := ItfProcessCollector;
Infeed.ProcessLinkedLists                 := ItfProcessList;
//-------------------------------------------------------------------------------------------------------------
// configure range of XtsStations for process
//
// see MAIN.StationParameterInit() for positions and dyn constraints
//-------------------------------------------------------------------------------------------------------------
ItfProcessCollector[Infeed.ProcessId].StationFirst        :=  1;
ItfProcessCollector[Infeed.ProcessId].StationLast         := 12;
//-------------------------------------------------------------------------------------------------------------
//-------------------------------------------------------------------------------------------------------------
//*************************************************************************************************************
//*************************************************************************************************************
// - BufferOutfeed  : single XtsStation which distributes movers to specified range 
//                    Infeed sends all movers here 
//                    BufferOutfeed ensures that OutputR2 and OutputR1 have 12 movers each for every job
//                    BufferOutfeed checks if the Queue of this single XtsStation is empty or not
//-------------------------------------------------------------------------------------------------------------
// whoami
//
// process target (Outfeed (OutfeedR2 & OutfeedR1) / 24 XtsStations)
//
//  - optional process target (Outfeed 12 XtsStations)
//-------------------------------------------------------------------------------------------------------------
_nBufferOutfeedTarget[1] := E_INSTANCE.OUTFEED_ROBOT_R1;
_nBufferOutfeedTarget[2] := E_INSTANCE.OUTFEED_ROBOT_R2;

BufferOutfeed.ProcessId              := E_INSTANCE.BUFFER_OUTFEED;
BufferOutfeed.ProcessTarget          := _nBufferOutfeedTarget; 
BufferOutfeed.CollectorInterface     := ItfProcessCollector;
BufferOutfeed.ProcessLinkedLists     := ItfProcessList;
//-------------------------------------------------------------------------------------------------------------
// configure range of XtsStations for process
//
// see MAIN.StationParameterInit() for positions and dyn constraints
//-------------------------------------------------------------------------------------------------------------
ItfProcessCollector[BufferOutfeed.ProcessId].StationFirst  := 25;
ItfProcessCollector[BufferOutfeed.ProcessId].StationLast   := 25;

_nStnFrst                                 := ProcessCollector[BufferOutfeed.ProcessId].StationFirst;
BufferOutfeed.CheckPosition          := 2500.0;
//-------------------------------------------------------------------------------------------------------------
//-------------------------------------------------------------------------------------------------------------
//*************************************************************************************************************
//*************************************************************************************************************
// - Outfeed_R1  : 12 XtsStations for Robot 
//                    All XtsStations must be filled before robot can start 
//                    affter process all movers are sent to Sender process (high speed for the way back)
//                     
//                    
//-------------------------------------------------------------------------------------------------------------
// whoami
//
// process target (SenderFast / 1 XtsStation)
//-------------------------------------------------------------------------------------------------------------
Outfeed_R1.ProcessId                      := E_INSTANCE.OUTFEED_ROBOT_R1;
Outfeed_R1.ProcessTarget                  := ProcessCollector[E_INSTANCE.SENDER_FAST].ProcessId;
Outfeed_R1.CollectorInterface             := ItfProcessCollector;
Outfeed_R1.ProcessLinkedLists             := ItfProcessList;
//-------------------------------------------------------------------------------------------------------------
// configure range of XtsStations for process
//
// see MAIN.StationParameterInit() for positions and dyn constraints
//-------------------------------------------------------------------------------------------------------------
ItfProcessCollector[Outfeed_R1.ProcessId].StationFirst  := 26;
ItfProcessCollector[Outfeed_R1.ProcessId].StationLast   := 37;

_nStnFrst                                 := ProcessCollector[Outfeed_R1.ProcessId].StationFirst;
Outfeed_R1.CheckPosition                  := 6000.0;
//-------------------------------------------------------------------------------------------------------------
//-------------------------------------------------------------------------------------------------------------
//*************************************************************************************************************
//*************************************************************************************************************
// - Outfeed_R2  : 12 XtsStations for Robot 
//                    All XtsStations must be filled before robot can start 
//                    affter process all movers are sent to Sender process (high speed for the way back)
//                     
//                    
//-------------------------------------------------------------------------------------------------------------
// whoami
//
// process target (SenderFast / 1 XtsStation)
//-------------------------------------------------------------------------------------------------------------
Outfeed_R2.ProcessId                      := E_INSTANCE.OUTFEED_ROBOT_R2;
Outfeed_R2.ProcessTarget                  := ProcessCollector[E_INSTANCE.SENDER_FAST].ProcessId;
Outfeed_R2.CollectorInterface             := ItfProcessCollector;
Outfeed_R2.ProcessLinkedLists             := ItfProcessList;
//-------------------------------------------------------------------------------------------------------------
// configure range of XtsStations for process
//
// see MAIN.StationParameterInit() for positions and dyn constraints
//-------------------------------------------------------------------------------------------------------------
ItfProcessCollector[Outfeed_R2.ProcessId].StationFirst  := 38;
ItfProcessCollector[Outfeed_R2.ProcessId].StationLast   := 49;

_nStnFrst                                 := ProcessCollector[Outfeed_R2.ProcessId].StationFirst;
Outfeed_R2.CheckPosition                  := 6000.0;
//-------------------------------------------------------------------------------------------------------------
//-------------------------------------------------------------------------------------------------------------
//*************************************************************************************************************
//*************************************************************************************************************
// - SenderFast  : 1 XtsStation 
//                    movers are handled when entering position area 
//                    movers are accelerated to max speed
//                    movers do not stop here
//                    
//-------------------------------------------------------------------------------------------------------------
// whoami
//
// process target (SenderBufferInfeed / 1 XtsStation)
//-------------------------------------------------------------------------------------------------------------
SenderFast.ProcessId                      := E_INSTANCE.SENDER_FAST;
SenderFast.ProcessTarget                  := ProcessCollector[E_INSTANCE.SENDER_BUFFER_INFEED].ProcessId;
SenderFast.CollectorInterface             := ItfProcessCollector;
SenderFast.ProcessLinkedLists             := ItfProcessList;
//-------------------------------------------------------------------------------------------------------------
// configure range of XtsStations for process
//
// see MAIN.StationParameterInit() for positions and dyn constraints
//-------------------------------------------------------------------------------------------------------------
ItfProcessCollector[SenderFast.ProcessId].StationFirst  := 51;
ItfProcessCollector[SenderFast.ProcessId].StationLast   := 51;

_nStnFrst                                 := ProcessCollector[SenderFast.ProcessId].StationFirst;
SenderFast.CheckPosition                  := GVL_XTS.StationParameter[_nStnFrst].rPosWait - 500.0;
//-------------------------------------------------------------------------------------------------------------
//-------------------------------------------------------------------------------------------------------------
//*************************************************************************************************************
//*************************************************************************************************************
// - SenderBufferInfeed  : 1 XtsStation 
//                    movers are handled when entering position area 
//                    movers are sent to BufferInfeed, so that BufferInfeed has 12 mover ready
//                    movers do stop here, wait until there is room for movers
//                    
//-------------------------------------------------------------------------------------------------------------
// whoami
//
// process target (SenderBufferInfeed / 1 XtsStation)
//-------------------------------------------------------------------------------------------------------------
SenderBufferInfeed.ProcessId              := E_INSTANCE.SENDER_BUFFER_INFEED;
SenderBufferInfeed.ProcessTarget          := ProcessCollector[E_INSTANCE.BUFFER_INFEED].ProcessId;
SenderBufferInfeed.CollectorInterface     := ItfProcessCollector;
SenderBufferInfeed.ProcessLinkedLists     := ItfProcessList;
//-------------------------------------------------------------------------------------------------------------
// configure range of XtsStations for process
//
// see MAIN.StationParameterInit() for positions and dyn constraints
//-------------------------------------------------------------------------------------------------------------
ItfProcessCollector[SenderBufferInfeed.ProcessId].StationFirst  := 52;
ItfProcessCollector[SenderBufferInfeed.ProcessId].StationLast   := 52;

_nStnFrst                                 := ProcessCollector[SenderBufferInfeed.ProcessId].StationFirst;
SenderBufferInfeed.CheckPosition          := GVL_XTS.StationParameter[_nStnFrst].rPosWait - 1250.0;
//-------------------------------------------------------------------------------------------------------------
//-------------------------------------------------------------------------------------------------------------
//*************************************************************************************************************

END_FUNCTION

// ---- APPLICATION/_Visu/SIM_TEST.TcVIS
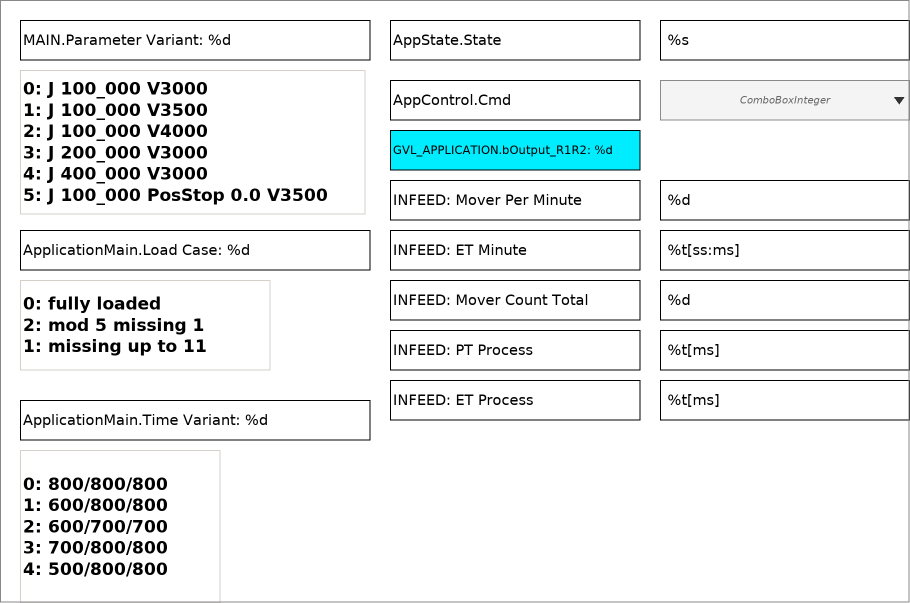
VISUALIZATION SIM_TEST  // 910x603
    Rectangle (20,230 350x40), "ApplicationMain.Load Case: %d", text variable: GVL_APPLICATION.ApplicationMain._nLoadCase
        OnMouseClick: write the text variable via VisuDialogs.Numpad, min 0, max 2
    Rectangle (20,400 350x40), "ApplicationMain.Time Variant: %d", text variable: GVL_APPLICATION.ApplicationMain._nTimeVariant
        OnMouseClick: write the text variable via VisuDialogs.Numpad, min 0, max 100
    Rectangle (20,20 350x40), "MAIN.Parameter Variant: %d", text variable: MAIN.nParameterVariant
        toggle MAIN.bWriteVariant
        OnMouseClick: write the text variable via VisuDialogs.Numpad, min 0, max 100
        OnMouseClick: execute { MAIN.bWriteVariant := TRUE; }
    Textfield (20,450 200x153), "0: 800/800/800 1: 600/800/800 2: 600/700/700 3: 700/800/800 4: 500/800/800"
    Textfield (20,280 250x90), "0: fully loaded 2: mod 5 missing 1 1: missing up to 11"
    Textfield (20,70 345x144), "0: J 100_000 V3000 1: J 100_000 V3500 2: J 100_000 V4000 3: J 200_000 V3000 4: J 400_000 V3000 5: J 100_000 PosStop 0.0 V3500"
    Rectangle (390,80 250x40), "AppControl.Cmd"
    ComboBoxInteger (660,80 250x40), variable: GVL_APPLICATION.AppControl.Cmd, text list: 'TL_E_INSTANCE_CMD'
    Rectangle (390,20 250x40), "AppState.State"
    Rectangle (660,20 250x40), "%s", text variable: GVL_APPLICATION.ApplicationMain._sAppState
    Rectangle (390,180 250x40), "INFEED: Mover Per Minute"
    Rectangle (660,180 250x40), "%d", text variable: GVL_APPLICATION.ProcessCollector[2]._AllStationMoverPerMinute
    Rectangle (390,280 250x40), "INFEED: Mover Count Total"
    Rectangle (660,280 250x40), "%d", text variable: GVL_APPLICATION.ProcessCollector[2]._nMoverCountTotal
    Rectangle (390,380 250x40), "INFEED: ET Process"
    Rectangle (660,380 250x40), "%t[ms]", text variable: GVL_APPLICATION.ApplicationMain._tonProcess[2].ET
    Rectangle (390,330 250x40), "INFEED: PT Process"
    Rectangle (660,330 250x40), "%t[ms]", text variable: GVL_APPLICATION.ApplicationMain._tProcess[2]
    Rectangle (390,230 250x40), "INFEED: ET Minute"
    Rectangle (660,230 250x40), "%t[ss:ms]", text variable: ProcessCollector[2]._tonPartsPerMinute.ET
    Rectangle (390,130 250x40), "GVL_APPLICATION.bOutput_R1R2: %d", text variable: GVL_APPLICATION.bOutput_R1R2, colour toggle: GVL_APPLICATION.bOutput_R1R2
        OnMouseClick: toggle GVL_APPLICATION.bOutput_R1R2
END_VISUALIZATION

// ---- GlobalTextList.TcGTLO
TEXTLIST GlobalTextList
  161 = ' %d'
  781 = ' %s'
  290 = ' %t[ms]'
  1009 = ' %t[ss:ms]'
  17 = ' STATION_ENABLE'
  34 = ' STATION_MOVER_ENTER'
  452 = ' STATION_MOVER_GONE'
  75 = ' STATION_MOVER_OUT'
  598 = ' STATION_PROCESS_DONE'
  750 = ' STATION_PROCESS_START'
  294 = '%.2f'
  191 = '%d'
  412 = '%r'
  836 = '%s'
  289 = '%t'
  343 = '0: 800/800/800'
  149 = '0: 800/800/800\n'
  77 = '0: 800/800/800\n1: 600/800/800'
  274 = '0: 800/800/800\n1: 600/800/800\n2: 600/700/700\n3: 700/800/800'
  1246 = '0: 800/800/800\n1: 600/800/800\n2: 600/700/700\n3: 700/800/800\n4: 500/800/800'
  605 = '0: fully loaded\n2: mod 5 missing 1\n1: missing up to 11'
  995 = '0: fully loaded\n2: mod 5 missing 1 1 = missing up to 11'
  232 = '0: J 100_000\n1: 600/800/800\n2: 600/700/700\n3: 700/800/800'
  450 = '0: J 100_000\n1: J 120_000\n2: J 160_000\n3: J 200_000\n4: J 400_000'
  960 = '0: J 100_000\n1: J 120_000\n2: J 160_000\n3: J 200_000\n4: J 400_000\n5: J 100_000 PosStop == 0.0'
  1159 = '0: J 100_000 V3000\n1: J 100_000 V3500\n2: J 100_000 V4000\n3: J 200_000 V3000\n4: J 400_000 V3000\n5: J 100_000 PosStop 0.0 V3500'
  129 = '0: J 100_000 V3000\n1: J 100_000 V3500\n2: J 100_000 V4000\n3: J 200_000 V3000\n4: J 400_000 V3000\n5: J 100_000 PosStop == 0.0 V3500'
  587 = '1: '
  248 = 'Activate'
  444 = 'Activate Visu list'
  704 = 'All Positions Valid'
  562 = 'AllAxisStanding'
  667 = 'AppControl.Cmd'
  32 = 'ApplicationMain.Load Case: %d'
  459 = 'ApplicationMain.Time Variant: %d'
  295 = 'AppState.State'
  878 = 'AxisCount Enabled: %d'
  162 = 'AxisCount: %d'
  516 = 'CA GroupInfo'
  914 = 'ConstantVelocity'
  929 = 'Control'
  707 = 'CyclicCheck: %s'
  660 = 'DC Link All Modules'
  359 = 'Decelerating'
  843 = 'Detected AxisCount: %d'
  243 = 'eDevice'
  244 = 'eSubdevice'
  242 = 'eType'
  772 = 'Expected AxisCount: %d'
  48 = 'GroupDisabled'
  915 = 'GroupError'
  495 = 'GroupErrorId: %d'
  975 = 'GroupErrorStop'
  940 = 'GroupHoming'
  300 = 'GroupMoving'
  807 = 'GroupNotReady'
  438 = 'GroupStandby'
  226 = 'GroupStatusBusy'
  204 = 'GroupStatusValid'
  973 = 'GroupStopping'
  180 = 'GVL_APPLICATION.bOutput_R1R2: %d'
  942 = 'GVL_XTS.CaGroupInfo'
  680 = 'ID Detection Active'
  238 = 'ID Detection Error'
  526 = 'ID Detection Mode: %s'
  29 = 'ID Detection Valid'
  245 = 'iErrorNumber'
  358 = 'INFEED: ET Minute'
  328 = 'INFEED: ET Process'
  268 = 'INFEED: Mover Count Total'
  682 = 'INFEED: Mover Per Minute'
  928 = 'INFEED: PT Process'
  211 = 'Info Act Pos Absolute'
  586 = 'Info Act Pos Modulo'
  21 = 'Info Mover Avoiding Collision'
  282 = 'Info Mover Coupled'
  398 = 'Info Mover Enabled'
  751 = 'Info Mover Error'
  907 = 'Info Mover Standstill'
  480 = 'Info nError ID'
  922 = 'Info Target Pos Absolute'
  16 = 'Info Target Pos Modulo'
  616 = 'InPosition'
  230 = 'Load Case'
  994 = 'Load Case %d'
  906 = 'MAIN.: %d'
  356 = 'MAIN.Parameter Variant: %d'
  713 = 'Mask: %b'
  972 = 'Mask: %d'
  779 = 'Mask: %s'
  726 = 'McGroupState:      %s'
  160 = 'McGroupState: %d  %s'
  974 = 'MOVER command'
  387 = 'Mover ID: %d'
  297 = 'Mover Position Assignement: %s'
  840 = 'MOVER result:  %s'
  53 = 'MOVER state:   %s'
  756 = 'nMoverSelected: %d'
  669 = 'nStation selected: %d'
  94 = 'Offset %.3f'
  427 = 'Offset: %.3f'
  312 = 'Operation Mode: %s'
  320 = 'Queue: %d'
  91 = 'Set Acceleration'
  399 = 'Set Delta'
  382 = 'Set Distance'
  757 = 'Set Gap'
  934 = 'Set Jerk'
  201 = 'Set Override'
  936 = 'Set Position'
  62 = 'Set Velocity'
  231 = 'State'
  748 = 'Station Control'
  267 = 'Station State'
  627 = 'STATION_ENABLE'
  247 = 'sText'
  54 = 'Target Station %d'
  567 = 'Target Station: %d'
  246 = 'tTime'
  517 = 'WRITE TO FILE'
  275 = 'XPU Command'
  227 = 'XpuResult:   %s'
  96 = 'XpuState:    %s'
  884 = 'XTS Station'
  572 = 'XTS Transport Check:  %s'
  212 = 'XTS Transport Check: %s'
  500 = 'XTS Transport Command'
  395 = 'XTS Transport Result: %s'
  798 = 'XTS Transport State:  %s'
  417 = 'XTS Transport State: %s'
END_TEXTLIST

// ---- XTS/_Visualization/STATION_VISU.TcVIS
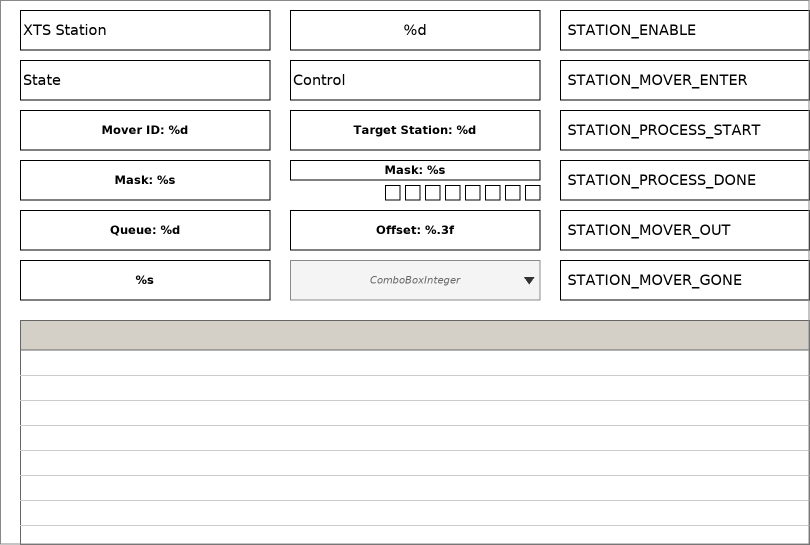
VISUALIZATION STATION_VISU  // 810x545
    Rectangle (20,10 250x40), "XTS Station"
    Rectangle (290,10 250x40), "%d", text variable: MAIN.nStationSelected
        OnMouseClick: write the text variable via VisuDialogs.Numpad, min 1, max MAX_STATION, title 'Selected Station'
    Rectangle (20,60 250x40), "State"
    Rectangle (290,60 250x40), "Control"
    Rectangle (20,210 250x40), "Queue: %d", text variable: GVL_XTS.StationState[MAIN.nStationSelected].nQueue
    Rectangle (20,110 250x40), "Mover ID: %d", text variable: GVL_XTS.StationState[MAIN.nStationSelected].nMoverId
    Rectangle (20,160 250x40), "Mask: %s", text variable: MAIN.sStationStateMask
    Rectangle (20,260 250x40), "%s", text variable: MAIN.sStationState
    ComboBoxInteger (290,260 250x40), variable: GVL_XTS.StationCtrl[MAIN.nStationSelected].eCmd, text list: 'TL_E_CTRL_STATION'
    Rectangle (290,210 250x40), "Offset: %.3f", text variable: GVL_XTS.StationCtrl[MAIN.nStationSelected].rOffset
    Rectangle (290,110 250x40), "Target Station: %d", text variable: GVL_XTS.StationCtrl[MAIN.nStationSelected].nTargetStation
        OnMouseClick: write the text variable via VisuDialogs.Numpad, min 1, max MAX_STATION, title 'Target Station'
    Rectangle (290,160 250x20), "Mask: %s", text variable: MAIN.sStationCtrlMask
    Rectangle (525,185 15x15)
        toggle GVL_XTS.StationCtrl[MAIN.nStationSelected].nMask.0
    Rectangle (505,185 15x15)
        toggle GVL_XTS.StationCtrl[MAIN.nStationSelected].nMask.1
    Rectangle (485,185 15x15)
        toggle GVL_XTS.StationCtrl[MAIN.nStationSelected].nMask.2
    Rectangle (465,185 15x15)
        toggle GVL_XTS.StationCtrl[MAIN.nStationSelected].nMask.3
    Rectangle (445,185 15x15)
        toggle GVL_XTS.StationCtrl[MAIN.nStationSelected].nMask.4
    Rectangle (425,185 15x15)
        toggle GVL_XTS.StationCtrl[MAIN.nStationSelected].nMask.5
    Rectangle (405,185 15x15)
        toggle GVL_XTS.StationCtrl[MAIN.nStationSelected].nMask.6
    Rectangle (385,185 15x15)
        toggle GVL_XTS.StationCtrl[MAIN.nStationSelected].nMask.7
    Rectangle (560,10 250x40), "STATION_ENABLE", colour toggle: MAIN.bStationEnable
        OnMouseClick: execute { GVL_XTS.StationCtrl[MAIN.nStationSelected].eCmd := E_STATION_CTRL.STATION_ENABLE; }
    Rectangle (560,60 250x40), "STATION_MOVER_ENTER", colour toggle: MAIN.bStationEnter
        OnMouseClick: execute { GVL_XTS.StationCtrl[MAIN.nStationSelected].eCmd := E_STATION_CTRL.STATION_MOVER_ENTER; }
    Rectangle (560,110 250x40), "STATION_PROCESS_START", colour toggle: MAIN.bStationStart
        OnMouseClick: execute { GVL_XTS.StationCtrl[MAIN.nStationSelected].eCmd := E_STATION_CTRL.STATION_PROCESS_START; }
    Rectangle (560,160 250x40), "STATION_PROCESS_DONE", colour toggle: MAIN.bStationDone
        OnMouseClick: execute { GVL_XTS.StationCtrl[MAIN.nStationSelected].eCmd := E_STATION_CTRL.STATION_PROCESS_DONE; }
    Rectangle (560,210 250x40), "STATION_MOVER_OUT", colour toggle: MAIN.bStationOut
        OnMouseClick: execute { GVL_XTS.StationCtrl[MAIN.nStationSelected].eCmd := E_STATION_CTRL.STATION_MOVER_OUT; }
    Rectangle (560,260 250x40), "STATION_MOVER_GONE", colour toggle: MAIN.bStationGone
        OnMouseClick: execute { GVL_XTS.StationCtrl[MAIN.nStationSelected].eCmd := E_STATION_CTRL.STATION_MOVER_GONE; }
    Table (20,320 790x225), data array: MAIN.tStationSelectedQueue
        p3854506369: MAIN.tStationSelectedQueue[INDEX].nMoverId
        p1892666644: MAIN.tStationSelectedQueue[INDEX].nTargetStation
        p338671338: MAIN.tStationSelectedQueue[INDEX].nMask
        p2170511999: MAIN.tStationSelectedQueue[INDEX].rOffset
END_VISUALIZATION

// ---- XTS/_Visualization/textlists/TL_E_CTRL_STATION.TcTLO
TEXTLIST TL_E_CTRL_STATION
  0 = 'STATION_CTRL_NULL'
  1 = 'STATION_INIT'
  10 = 'STATION_DISABLE'
  11 = 'STATION_ENABLE'
  20 = 'STATION_MOVER_ENTER'
  21 = 'STATION_MOVER_ENTER_RETRY'
  22 = 'STATION_MOVER_SEND'
  30 = 'STATION_PROCESS_START'
  31 = 'STATION_PROCESS_DONE'
  50 = 'STATION_MOVER_OUT'
  51 = 'STATION_MOVER_OUT_RETRY'
  60 = 'STATION_MOVER_GONE'
   = ''
END_TEXTLIST

// ---- XTS/_Visualization/XTS_TRANSPORT.TcVIS
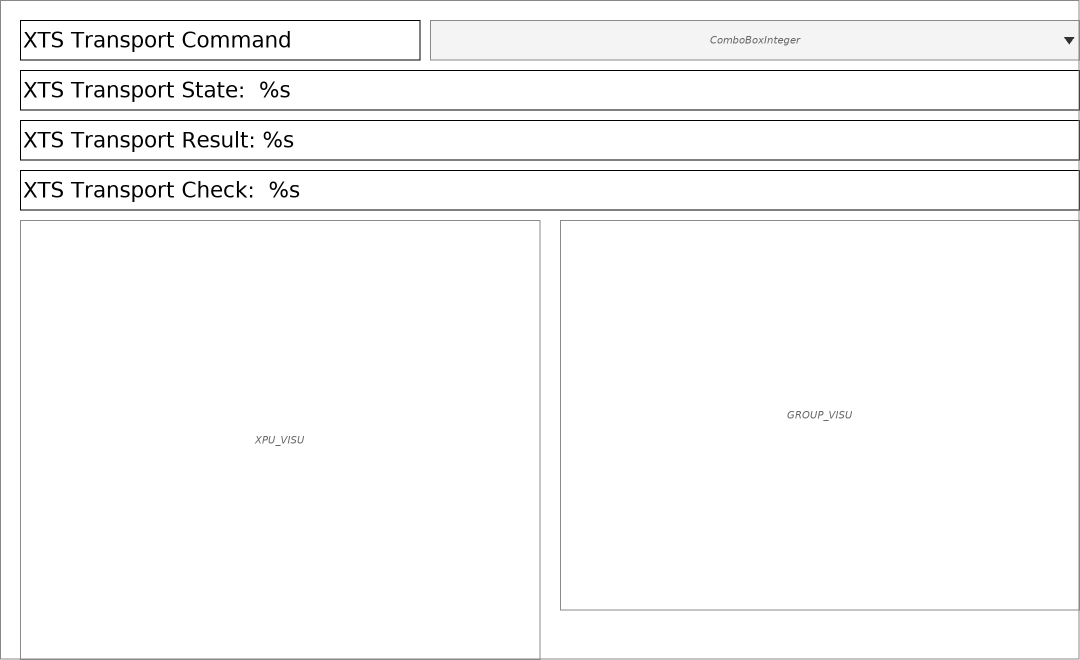
VISUALIZATION XTS_TRANSPORT  // 1080x660
    Rectangle (20,20 400x40), "XTS Transport Command"
    ComboBoxInteger (430,20 650x40), variable: GVL_XTS.XtsTransportCtrl.Cmd, text list: 'TL_E_CTRL_TRANSPORT'
    Rectangle (20,70 1060x40), "XTS Transport State: %s", text variable: MAIN.sTransportState
    Rectangle (20,120 1060x40), "XTS Transport Result: %s", text variable: MAIN.sTransportResult
    Rectangle (20,170 1060x40), "XTS Transport Check: %s", text variable: MAIN.sTransportCheck
    Frame (20,220 520x440)
        shows XPU_VISU(stXpuState := GVL_XTS.XtsTransportState.XpuState, stXpuInfo := GVL_XTS.XtsTransportState.XpuInfo, stXpuStrings := MAIN.stXpuStrings)
    Frame (560,220 520x390)
        shows GROUP_VISU(stGroupInfo := GVL_XTS.XtsTransportState.GroupInfo, sGroupState := MAIN.sCaGroupState)
END_VISUALIZATION
